# EPICS alarm handler configuration: mps_database/bare/alarms/areas/mpln_ltus_mp03.alhConfig
GROUP NULL MPLN:LTUS:MP03:1
$ALIAS MPS Link Node 205
$GUIDANCE
LTUH MPS
   Group Name: MPLN:LTUS:MP03:1
   Summary PV:  MPLN:LTUS:MP03:1:STATSUMY
$END
CHANNEL  MPLN:LTUS:MP03:1    MPLN:LTUS:MP03:1:MPS_EN_RBV		-----
CHANNEL  MPLN:LTUS:MP03:1    MPLN:LTUS:MP03:1:LC1_MODE_RBV		-----
